INTERFACE ITF_EM_Transport

METHOD Abort : BOOL
VAR_INPUT
END_VAR
END_METHOD

PROPERTY Auto : BOOL
GET
END_GET
SET
END_SET
END_PROPERTY

PROPERTY Manueel : BOOL
GET
END_GET
SET
END_SET
END_PROPERTY

METHOD Reset : BOOL
VAR_INPUT
END_VAR
END_METHOD

PROPERTY RPM : INT
GET
END_GET
SET
END_SET
END_PROPERTY

METHOD Start : BOOL
VAR_INPUT
END_VAR
END_METHOD

PROPERTY State : E_State_PackML
GET
END_GET
END_PROPERTY

METHOD Stop : BOOL
VAR_INPUT
END_VAR
END_METHOD

PROPERTY Tag : STRING
GET
END_GET
END_PROPERTY

METHOD ZeroAllVar : BOOL
VAR_INPUT
END_VAR
END_METHOD

END_INTERFACE

(* stored: Version 1.1.0.1, ProductVersion 3.1.4024.12
   Itf ITF_EM_Transport: Id {31841963-59b9-4495-8c67-f6cc39e2ec03}
   Folder Methods: Id {13a2a41d-5965-4014-8648-897ab3557794}
   Folder Properties: Id {6d943727-7254-448b-b0cd-a158dfcfefa0}
   Method Abort: Id {5e1801f7-a3ec-4e4c-a24c-84c34413db12}
   Property Auto: Id {fc6e3e21-26ef-42cc-a0a1-4e367a1afd38}
   Get Get: Id {a8e83ab7-d955-4f17-af6b-b4f91749c03c}
   Set Set: Id {f4508969-96e8-47e0-8db1-9dac65f8a78b}
   Property Manueel: Id {6ead2dc1-40a7-4622-b37c-8156eff25637}
   Get Get: Id {d727bb69-932e-4891-beab-4685030f0244}
   Set Set: Id {f3764319-7ed6-4936-8759-d79ec55acae6}
   Method Reset: Id {76be5b52-adde-42a0-a2a7-2b49f3338760}
   Property RPM: Id {eb6f6ce5-4e0f-42a0-bd35-cb3c4017b1c7}
   Get Get: Id {7bd33afd-0915-4944-bf5a-cc2e3fb422b1}
   Set Set: Id {492f15b3-6398-40e2-b61a-6dcf52b945ab}
   Method Start: Id {35f1ec48-e4bc-4cbe-8559-7a1414d56cd7}
   Property State: Id {3684ca1a-131e-4664-b674-ec6ee3bc6967}
   Get Get: Id {67689f73-1d16-4394-8faa-139d23b6137f}
   Method Stop: Id {e374a9c2-6372-468d-96a4-db90f40a1bfb}
   Property Tag: Id {ddfe14d4-3f8a-4340-b285-9dedd437d792}
   Get Get: Id {8bca3ec6-a0ee-45c1-9283-d6f64f1af812}
   Method ZeroAllVar: Id {cd71b208-4c45-4038-bac7-7767f90dc3d7} *)
